FUNCTION_BLOCK FB_CreatePartProgram 
VAR_INPUT
	Execute 	: BOOL;
	sData		: STRING(8191);
	sNetId		: STRING;
	sPathName	: STRING;
END_VAR
VAR_OUTPUT
	Busy : BOOL;
	Done : BOOL;
	Error : BOOL;
	ErrorID : DINT;
	ErrorSubID : UDINT;
	Q_tElapsedTime	: TIME;
END_VAR
VAR
	iState : DINT := -1;
	fbFileOpen: FB_FileOpen;
	fbFileClose: FB_FileClose;
	fbFileWrite: FB_FileWrite;
	hSrcFile : UINT;
	RTRIG_Execute : R_TRIG;
	TON_TimeElapsed : TON;
	TON_Timeout		: TON;
END_VAR

TON_Timeout(IN := Busy, PT := T#20S);
IF TON_Timeout.Q THEN
	
	iState := 1999;
END_IF

RTRIG_Execute(CLK := Execute);
TON_TimeElapsed(PT:= T#5S);
IF(RTRIG_Execute.Q) THEN
	ErrorID := 0;
	ErrorSubID := 0;
	
	iState := 0;
ELSIF NOT Execute AND NOT Busy THEN
	Busy			:= FALSE;
	Done			:= FALSE;
	Error			:= FALSE;
	
	iState := -1;
END_IF

CASE iState OF
	-1:
		;
	0:
		TON_TimeElapsed.IN := TRUE;
		fbFileOpen.bExecute := TRUE;
		Busy := TRUE;
		iState := 10;
			
	10:
        fbFileOpen.bExecute := FALSE; 
        IF NOT fbFileOpen.bBusy THEN 
        	IF fbFileOpen.bError THEN 
            	ErrorSubID := fbFileOpen.nErrId; 
                iState := 1010;
               ELSE 
                    hSrcFile := fbFileOpen.hFile;
					fbFileWrite.bExecute := TRUE; 
                 	iState := 20;
               END_IF 
          END_IF
		  
	20:
          fbFileWrite.bExecute := FALSE; 
          IF NOT fbFileWrite.bBusy THEN 
               IF fbFileWrite.bError THEN 
                    ErrorSubID := fbFileWrite.nErrId; 
                    iState := 1020;
               ELSE 
				   fbFileClose.bExecute := TRUE;
				   
                   iState := 30;
               END_IF 
          END_IF

	30:
		 fbFileClose.bExecute := FALSE;
		 IF NOT fbFileClose.bBusy THEN 
         	IF fbFileClose.bError THEN 
            	ErrorSubID := TO_DINT(fbFileClose.nErrId);  
            END_IF 
           
			Q_tElapsedTime 		:= TON_TimeElapsed.ET;
			
			TON_TimeElapsed.IN 	:= FALSE;
			
			iState 				:= 999;
          END_IF 

	999:
			Busy	 			:= FALSE;
			Done				:= TRUE;
		
END_CASE

IF(iState > 999 OR TON_TimeElapsed.Q) THEN
	Error 	:= TRUE;
	ErrorID := iState;
	Busy 	:= FALSE;
ELSE
	Error := FALSE;
END_IF

A_Call();

ACTION A_Call:
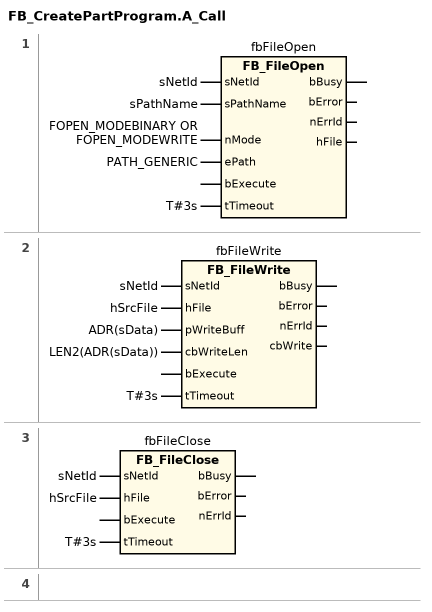
// NETWORK 1
fbFileOpen(
    sNetId := sNetId,
    sPathName := sPathName,
    nMode := FOPEN_MODEBINARY OR FOPEN_MODEWRITE,
    ePath := PATH_GENERIC,
    tTimeout := T#3s); // FB_FileOpen

// NETWORK 2
fbFileWrite(
    sNetId := sNetId,
    hFile := hSrcFile,
    pWriteBuff := ADR(sData),
    cbWriteLen := LEN2(ADR(sData)),
    tTimeout := T#3s); // FB_FileWrite

// NETWORK 3
fbFileClose(sNetId := sNetId, hFile := hSrcFile, tTimeout := T#3s); // FB_FileClose

// NETWORK 4
END_ACTION

END_FUNCTION_BLOCK

(* stored: Version 1.1.0.1, ProductVersion 3.1.4024.13
   POU FB_CreatePartProgram: Id {627b290a-a58f-4ab5-b7aa-cfbc324fdea6}, SpecialFunc None
   Action A_Call: Id {5a4a29d0-1260-4593-9792-71bf7a2dfc20} *)
